{attribute 'qualified_only'}
{attribute 'strict'}
{attribute 'to_string'}
TYPE E_STATION_TYPE :
(
	INVALID,
  STATION_PROCESS,      // default station with/without process
  STATION_GEAR_IN_POS   // GearInPos station for flying saw with MasterAxis
)USINT;
END_TYPE

(* stored: Version 1.1.0.1
   DUT E_STATION_TYPE: Id {2d05881f-2e7a-4331-ae1b-744610f5b5cb} *)
